// LS Electric XG5000 project: jg1
// PLC NewPLC
// module base 0 slot 0: 입출력 모듈:XBM-DN32H (DC 24V입력/TR 출력, 32점)

PROGRAM NewProgram (task: 스캔 프로그램)

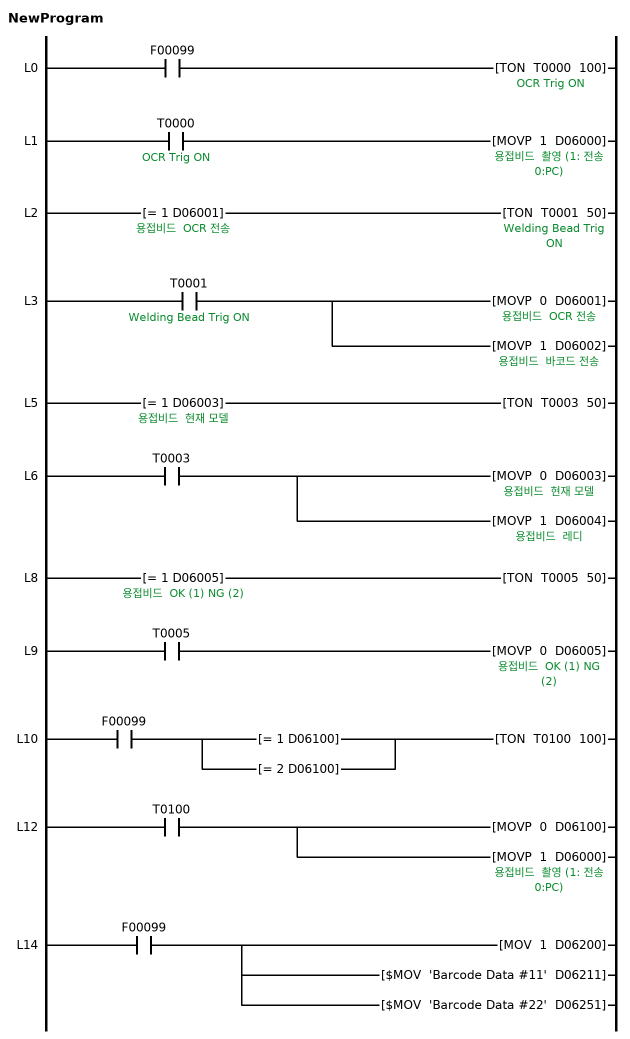
; L0
LOAD      F00099
TON       T0000 100	// OCR Trig ON
; L1
LOAD      T0000	// OCR Trig ON
MOVP      1 D06000	// 용접비드  촬영 (1: 전송 0:PC)
; L2
LOAD=     1 D06001	// 용접비드  OCR 전송
TON       T0001 50	// Welding Bead Trig ON
; L3
LOAD      T0001	// Welding Bead Trig ON
MOVP      0 D06001	// 용접비드  OCR 전송
MOVP      1 D06002	// 용접비드  바코드 전송
; L5
LOAD=     1 D06003	// 용접비드  현재 모델
TON       T0003 50
; L6
LOAD      T0003
MOVP      0 D06003	// 용접비드  현재 모델
MOVP      1 D06004	// 용접비드  레디 
; L8
LOAD=     1 D06005	// 용접비드  OK (1) NG (2)
TON       T0005 50
; L9
LOAD      T0005
MOVP      0 D06005	// 용접비드  OK (1) NG (2)
; L10
LOAD      F00099
LOAD=     1 D06100
OR=       2 D06100
AND LOAD
TON       T0100 100
; L12
LOAD      T0100
MOVP      0 D06100
MOVP      1 D06000	// 용접비드  촬영 (1: 전송 0:PC)
; L14
LOAD      F00099
MOV       1 D06200
$MOV      'Barcode Data #11' D06211
$MOV      'Barcode Data #22' D06251

VARIABLES AND COMMENTS (devices not used above)
K00591	BIT	CAR TYPE TMA 2WD
K00592	BIT	CAR TYPE TMA 4WD
K00593	BIT	CAR TYPE ON 2WD
K00594	BIT	CAR TYPE ON 4WD
T0010	BIT/WORD	Vision Ready
T0002	BIT/WORD	Trig OFF
P00020	BIT	OCR Trig
P00021	BIT	Visin Trig
D06010	WORD	용접비드  OCR DATA #1
D06011	WORD	용접비드  OCR DATA #2
D06012	WORD	용접비드  OCR DATA #3
D06013	WORD	용접비드  OCR DATA #4
D06020	WORD	용접비드  바코드 #1
T0020	BIT/WORD	Alive Alarm
K00600	BIT	Camera End
D04010	WORD	용접 비드 OCR
D04020	WORD	용접 바코드